{attribute 'linkalways'} 
{attribute 'no_explicit_call' := 'This FB is a CLASS and must be accessed using methods or properties'}
{attribute 'enable_dynamic_creation'}
FUNCTION_BLOCK Node_ContainerType_Vector_TcVnPoint2_REAL EXTENDS Node
VAR
    out : _GUID;
END_VAR

METHOD PUBLIC  Clone : I_Node
VAR
	pNode : POINTER TO Node_ContainerType_Vector_TcVnPoint2_REAL;
END_VAR
pNode := __NEW(Node_ContainerType_Vector_TcVnPoint2_REAL);
Clone := pNode^;
END_METHOD

METHOD FB_init : BOOL
VAR_INPUT
	bInitRetains : BOOL; // if TRUE, the retain variables are initialized (warm start / cold start)
	bInCopyCode : BOOL;  // if TRUE, the instance afterwards gets moved into the copy code (online change)
END_VAR
AddOutput('out', out);
END_METHOD

METHOD PROTECTED OnExecute
out.Value := ContainerType_Vector_TcVnPoint2_REAL;
END_METHOD

END_FUNCTION_BLOCK

(* stored: Version 1.1.0.1, ProductVersion 3.1.4026.17
   POU Node_ContainerType_Vector_TcVnPoint2_REAL: Id {5c6212ef-0fdb-0d14-1469-c990e33c44fe}, SpecialFunc None
   Folder Constructor: Id {c249c59e-7abe-0308-28d3-d840de8a574f}
   Method Clone: Id {417b9648-41f9-009c-107f-ba3476349c11}
   Method FB_init: Id {77afaa0b-a75e-0534-325b-ab57f7e8d505}
   Method OnExecute: Id {dbe2de08-ee5b-094f-039d-07c2f086b7d2} *)
